{attribute 'GeneratedUsingTerminal: EK1122-0000-0018'}
{attribute addProperty BoxType "EK1122-0000-0018"}
{attribute addProperty Id "Beckhoff_EL31xxsub_EK1100EK1100_1FC0878B2"}
{attribute addProperty CRC "406529280"}
{attribute addProperty Size "2"}
TYPE Beckhoff_EL31xxEK1122_183B2500 EXTENDS EK1122_1FC0878B :
STRUCT
	{attribute addProperty Name "Beckhoff_EL31xxsub_EK1100"}
	{attribute addProperty PreviousPort "Beckhoff EL31xxEK1122 : D"}
	Beckhoff_EL31xxsub_EK1100 : EK1100_1FC0878B;
END_STRUCT
END_TYPE

(* stored: Version 1.2.0.0, ProductVersion 3.1.4024.9
   DUT Beckhoff_EL31xxEK1122_183B2500: Id {e08faaf6-0d47-493b-93a6-cf54b7bcfc51} *)
